Omron CX-Programmer project NuevoProyecto (CX-Programmer 9.54)

# PLC NuevoPLC1: CJ2M CPU31

## Program NuevoPrograma1 (cyclic task 0)
Local symbols
Entrada1 0.00 BOOL
Entrada15 0.14 BOOL
Entrada16 0.15 BOOL
Entrada2 0.01 BOOL
Entrada3 0.02 BOOL
Entrada4 0.03 BOOL
Entrada5 0.04 BOOL
Entrada6 0.05 BOOL
Entrada7 0.06 BOOL
Entrada8 0.07 BOOL
Entrada9 0.08 BOOL
FCNH BOOL
GYUK BOOL
Intermitente 0.11 BOOL
P_on BOOL
Salida1 1.00 BOOL
Salida11 1.10 BOOL
Salida12 1.11 BOOL
Salida13 1.12 BOOL
Salida14 1.13 BOOL
Salida15 1.14 BOOL
Salida16 1.15 BOOL
Salida2 1.01 BOOL
Salida3 1.02 BOOL
Salida4 1.03 BOOL
Salida5 1.04 BOOL
Salida6 1.05 BOOL
Salida7 1.06 BOOL
Salida8 1.07 BOOL
Salida9 1.08 BOOL
VHULK BOOL

### Section Sección1

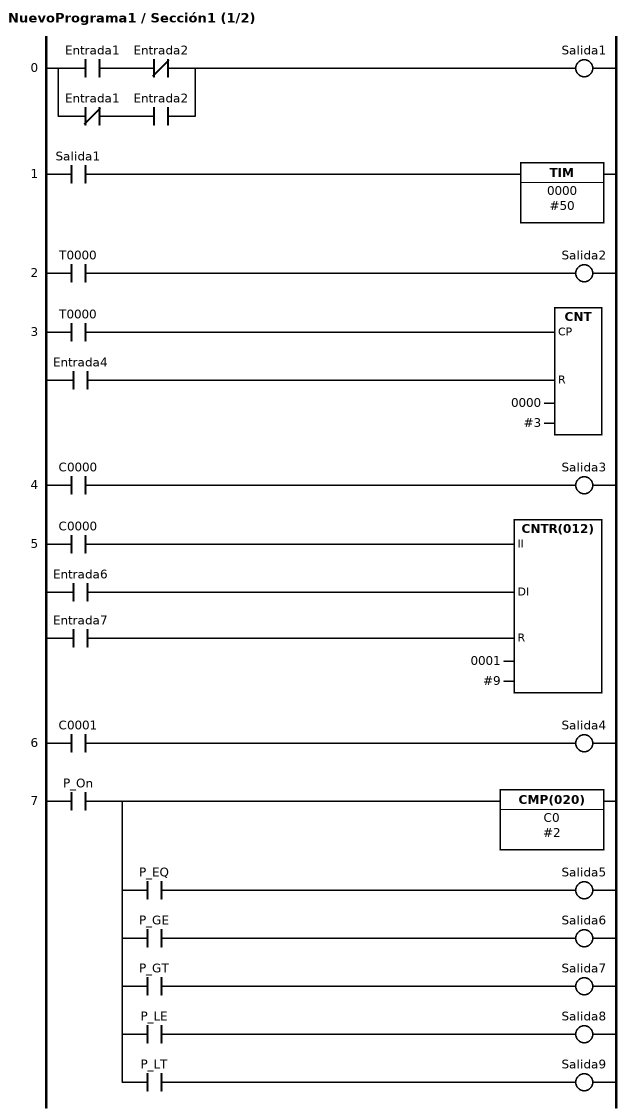
; rung 0
LD Entrada1
ANDNOT Entrada2
LDNOT Entrada1
AND Entrada2
ORLD
OUT Salida1
; rung 1
LD Salida1
TIM 0000 #50
; rung 2
LD T0000
OUT Salida2
; rung 3
LD T0000
LD Entrada4
CNT 0000 #3
; rung 4
LD C0000
OUT Salida3
; rung 5
LD C0000
LD Entrada6
LD Entrada7
CNTR(012) 0001 #9
; rung 6
LD C0001
OUT Salida4
; rung 7
LD P_On
OUT TR0
CMP(020) C0 #2
AND P_EQ
OUT Salida5
LD TR0
AND P_GE
OUT Salida6
LD TR0
AND P_GT
OUT Salida7
LD TR0
AND P_LE
OUT Salida8
LD TR0
AND P_LT
OUT Salida9

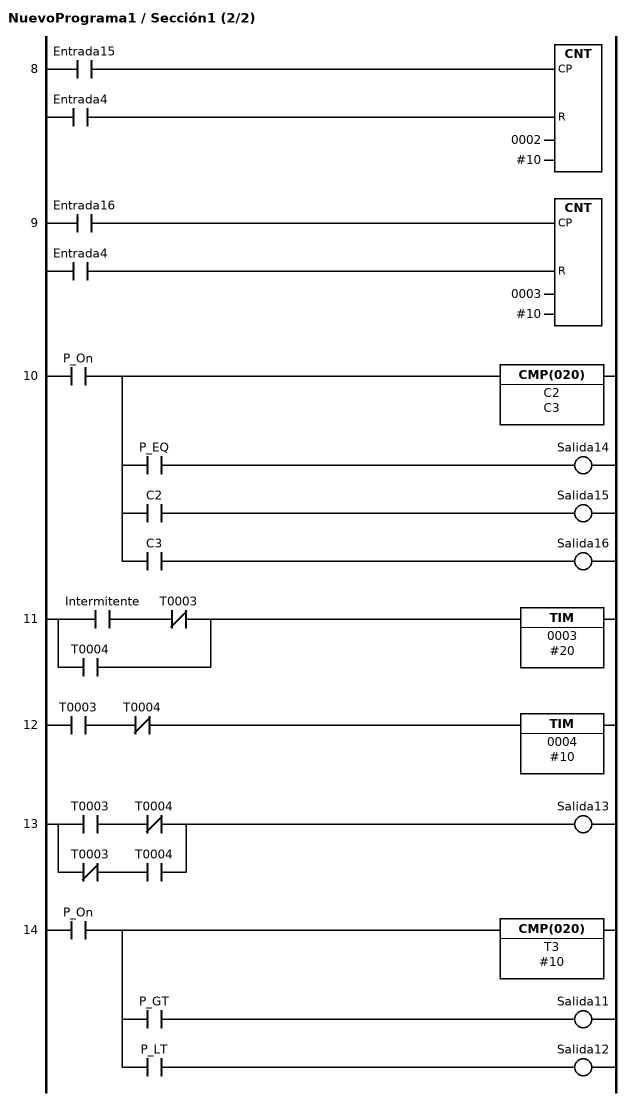
; rung 8
LD Entrada15
LD Entrada4
CNT 0002 #10
; rung 9
LD Entrada16
LD Entrada4
CNT 0003 #10
; rung 10
LD P_On
OUT TR0
CMP(020) C2 C3
AND P_EQ
OUT Salida14
LD TR0
AND C2 #0
OUT Salida15
LD TR0
AND C3 #0
OUT Salida16
; rung 11
LD Intermitente
ANDNOT T0003
OR T0004
TIM 0003 #20
; rung 12
LD T0003
ANDNOT T0004
TIM 0004 #10
; rung 13
LD T0003
ANDNOT T0004
LDNOT T0003
AND T0004
ORLD
OUT Salida13
; rung 14
LD P_On
OUT TR0
CMP(020) T3 #10
AND P_GT
OUT Salida11
LD TR0
AND P_LT
OUT Salida12

### Section END
; rung 0
END(001)